(* CODESYS project BagFeedMotorIMove.Traverse_active.xml

Project tree, tasks and I/O mapping:
*)

// Traverse_active
ACTION Traverse_active:
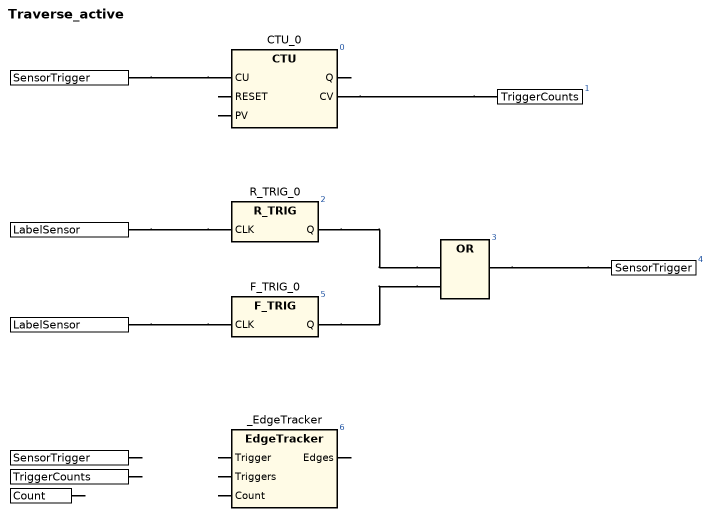
CTU_0(CU := SensorTrigger); // CTU
TriggerCounts := CTU_0.CV;
R_TRIG_0(CLK := LabelSensor); // R_TRIG
SensorTrigger := R_TRIG_0.Q OR F_TRIG_0.Q;
F_TRIG_0(CLK := LabelSensor); // F_TRIG
_EdgeTracker(); // EdgeTracker
// SensorTrigger: input not connected
// TriggerCounts: input not connected
// Count: input not connected
END_ACTION
